// LS Electric XG5000 project: 동남137
// PLC NewPLC
// module base 0 slot 0: 입출력 모듈:XBC-DN/DP14E (DC 24V 입력 8점, 트랜지스터 출력 6점)

PROGRAM NewProgram (task: 스캔 프로그램)

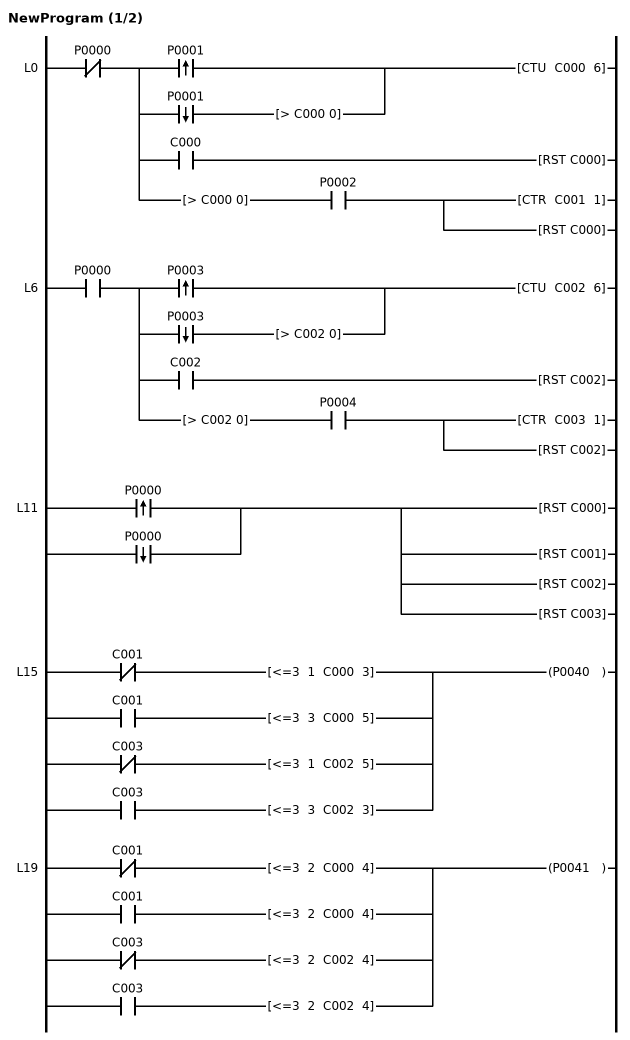
; L0
LOAD NOT  P0000
MPUSH
LOADP     P0001
LOADN     P0001
AND>      C000 0
OR LOAD
AND LOAD
CTU       C000 6
MLOAD
AND       C000
RST       C000
MPOP
AND>      C000 0
AND       P0002
CTR       C001 1
RST       C000
; L6
LOAD      P0000
MPUSH
LOADP     P0003
LOADN     P0003
AND>      C002 0
OR LOAD
AND LOAD
CTU       C002 6
MLOAD
AND       C002
RST       C002
MPOP
AND>      C002 0
AND       P0004
CTR       C003 1
RST       C002
; L11
LOADP     P0000
ORN       P0000
RST       C000
RST       C001
RST       C002
RST       C003
; L15
LOAD NOT  C001
AND<=3    1 C000 3
LOAD      C001
AND<=3    3 C000 5
OR LOAD
LOAD NOT  C003
AND<=3    1 C002 5
OR LOAD
LOAD      C003
AND<=3    3 C002 3
OR LOAD
OUT       P0040
; L19
LOAD NOT  C001
AND<=3    2 C000 4
LOAD      C001
AND<=3    2 C000 4
OR LOAD
LOAD NOT  C003
AND<=3    2 C002 4
OR LOAD
LOAD      C003
AND<=3    2 C002 4
OR LOAD
OUT       P0041

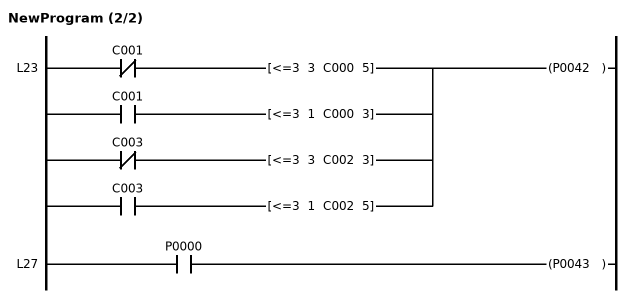
; L23
LOAD NOT  C001
AND<=3    3 C000 5
LOAD      C001
AND<=3    1 C000 3
OR LOAD
LOAD NOT  C003
AND<=3    3 C002 3
OR LOAD
LOAD      C003
AND<=3    1 C002 5
OR LOAD
OUT       P0042
; L27
LOAD      P0000
OUT       P0043